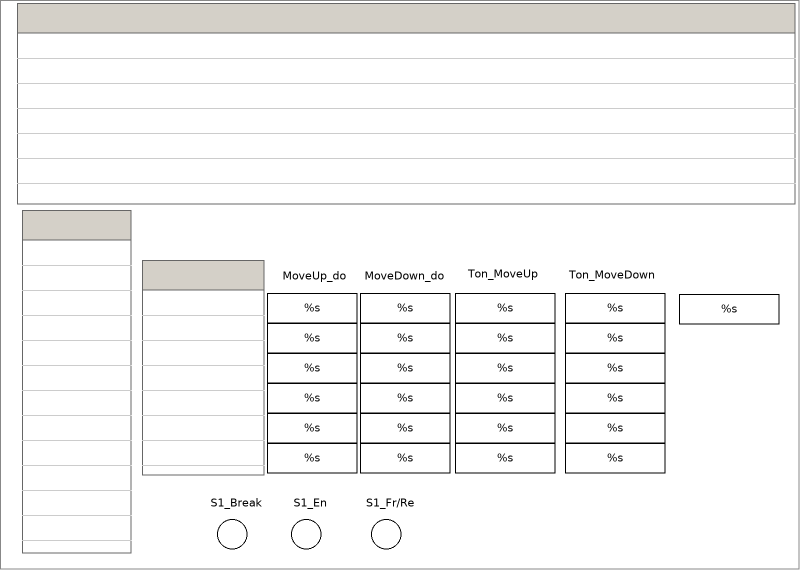
VISUALIZATION VIS_UpDownSlot  // 800x570
    Table (17,3 778x201), data array: GVL_API.stUpDownSlot
        p3854506369: GVL_API.stUpDownSlot[INDEX].error_code
        p1892666644: GVL_API.stUpDownSlot[INDEX].state
        p338671338: GVL_API.stUpDownSlot[INDEX].sensor_up
        p2170511999: GVL_API.stUpDownSlot[INDEX].sensor_down
        p3723444502: GVL_API.stUpDownSlot[INDEX].Error
        p1218418051: GVL_API.stUpDownSlot[INDEX].Initialize
        p746581629: GVL_API.stUpDownSlot[INDEX].MoveDown
        p3104783080: GVL_API.stUpDownSlot[INDEX].MoveUp
        p2501879983: GVL_API.stUpDownSlot[INDEX].Setoff
        p7306298: GVL_API.stUpDownSlot[INDEX].timeout_up
        p1933151965: GVL_API.stUpDownSlot[INDEX].timeout_down
        p3863566920: GVL_API.stUpDownSlot[INDEX].extra_down_time
        p4242324053: extra_time
        Columns.Column.[8].Template: toggle GVL_API.stUpDownSlot[INDEX].Setoff
        Columns.Column.[6].Template: toggle GVL_API.stUpDownSlot[INDEX].MoveDown
        Columns.Column.[10].Template: OnMouseDown: write GVL_API.stUpDownSlot[INDEX].timeout_down via Default
        Columns.Column.[5].Template: toggle GVL_API.stUpDownSlot[INDEX].Initialize
        Columns.Column.[11].Template: OnMouseDown: write GVL_API.stUpDownSlot[INDEX].extra_down_time via Default
        Columns.Column.[7].Template: toggle GVL_API.stUpDownSlot[INDEX].MoveUp
        Columns.Column.[9].Template: OnMouseDown: write GVL_API.stUpDownSlot[INDEX].timeout_up via Default
        Columns.Column.[1].Template: GVL_API.stUpDownSlot[INDEX].state=100
    Rectangle (565,293 100x30), "%s", text variable: P_UpDownSlot.UpDownSlot_S1.Ton_MoveDown_do.ET
    Table (142,260 122x215), data array: stInput.biUDS_sensor_up_S
        p1892666644: stInput.biUDS_sensor[INDEX].sensor_up_right
        p338671338: stInput.biUDS_sensor[INDEX].sensor_down_left
        p2170511999: stInput.biUDS_sensor[INDEX].sensor_down_right
        p3854506369: stInput.biUDS_sensor_up_S[INDEX]
        Columns.Column.[0].Template: toggle stInput.biUDS_sensor_up_S[INDEX]
    Rectangle (565,353 100x30), "%s", text variable: P_UpDownSlot.UpDownSlot_S2_S6[3].Ton_MoveDown_do.ET
    Rectangle (565,383 100x30), "%s", text variable: P_UpDownSlot.UpDownSlot_S2_S6[4].Ton_MoveDown_do.ET
    Rectangle (565,413 100x30), "%s", text variable: P_UpDownSlot.UpDownSlot_S2_S6[5].Ton_MoveDown_do.ET
    Rectangle (565,323 100x30), "%s", text variable: P_UpDownSlot.UpDownSlot_S2_S6[2].Ton_MoveDown_do.ET
    Rectangle (455,293 100x30), "%s", text variable: P_UpDownSlot.UpDownSlot_S1.Ton_MoveUp_do.ET
    Rectangle (455,323 100x30), "%s", text variable: P_UpDownSlot.UpDownSlot_S2_S6[2].Ton_MoveUp_do.ET
    Rectangle (455,353 100x30), "%s", text variable: P_UpDownSlot.UpDownSlot_S2_S6[3].Ton_MoveUp_do.ET
    Rectangle (455,383 100x30), "%s", text variable: P_UpDownSlot.UpDownSlot_S2_S6[4].Ton_MoveUp_do.ET
    Rectangle (455,413 100x30), "%s", text variable: P_UpDownSlot.UpDownSlot_S2_S6[5].Ton_MoveUp_do.ET
    Label (559,260 106x30), "Ton_MoveDown"
    Label (451,259 104x30), "Ton_MoveUp"
    Table (22,210 109x343), data array: stInput.biUDS_sensor_down_S1
        p3854506369: stInput.biUDS_sensor_down_S1[INDEX]
        p1892666644: stInput.biUDS_sensor[INDEX].sensor_up_right
        p338671338: stInput.biUDS_sensor[INDEX].sensor_down_left
        p2170511999: stInput.biUDS_sensor[INDEX].sensor_down_right
        Columns.Column.[0].Template: toggle stInput.biUDS_sensor_down_S1[INDEX]
    Rectangle (565,443 100x30), "%s", text variable: P_UpDownSlot.UpDownSlot_S2_S6[6].Ton_MoveDown_do.ET
    Rectangle (455,443 100x30), "%s", text variable: P_UpDownSlot.UpDownSlot_S2_S6[6].Ton_MoveUp_do.ET
    Rectangle (679,294 100x30), "%s", text variable: P_UpDownSlot.UpDownSlot_S1.Ton_MoveDown_delay_do.ET
    Ellipse (217,519 30x30), colour toggle: stOutput.bqS1_Break
    Label (202,488 69x30), "S1_Break"
    Rectangle (267,323 90x30), "%s", text variable: stOutput.bqUDS_MoveUp_do[2], colour toggle: stOutput.bqUDS_MoveUp_do[2]
    Label (268,261 93x30), "MoveUp_do"
    Rectangle (360,323 90x30), "%s", text variable: stOutput.bqUDS_MoveDown_do[2], colour toggle: stOutput.bqUDS_MoveDown_do[2]
    Label (358,261 93x30), "MoveDown_do"
    Rectangle (267,353 90x30), "%s", text variable: stOutput.bqUDS_MoveUp_do[3], colour toggle: stOutput.bqUDS_MoveUp_do[3]
    Rectangle (267,383 90x30), "%s", text variable: stOutput.bqUDS_MoveUp_do[4], colour toggle: stOutput.bqUDS_MoveUp_do[4]
    Rectangle (267,413 90x30), "%s", text variable: stOutput.bqUDS_MoveUp_do[5], colour toggle: stOutput.bqUDS_MoveUp_do[5]
    Rectangle (267,443 90x30), "%s", text variable: stOutput.bqUDS_MoveUp_do[6], colour toggle: stOutput.bqUDS_MoveUp_do[6]
    Rectangle (360,353 90x30), "%s", text variable: stOutput.bqUDS_MoveDown_do[3], colour toggle: stOutput.bqUDS_MoveDown_do[3]
    Rectangle (360,383 90x30), "%s", text variable: stOutput.bqUDS_MoveDown_do[4], colour toggle: stOutput.bqUDS_MoveDown_do[4]
    Rectangle (360,413 90x30), "%s", text variable: stOutput.bqUDS_MoveDown_do[5], colour toggle: stOutput.bqUDS_MoveDown_do[5]
    Rectangle (360,443 90x30), "%s", text variable: stOutput.bqUDS_MoveDown_do[6], colour toggle: stOutput.bqUDS_MoveDown_do[6]
    Rectangle (267,293 90x30), "%s", text variable: P_UpDownSlot.UpDownSlot_S1.MoveUp_do, colour toggle: P_UpDownSlot.UpDownSlot_S1.MoveUp_do
    Rectangle (360,293 90x30), "%s", text variable: P_UpDownSlot.UpDownSlot_S1.MoveDown_do, colour toggle: P_UpDownSlot.UpDownSlot_S1.MoveDown_do
    Ellipse (291,519 30x30), colour toggle: stOutput.bqS1_Drive_enabled
    Label (276,488 69x30), "S1_En"
    Ellipse (371,519 30x30), colour toggle: stOutput.bqS1_Forward_Reverse
    Label (356,488 69x30), "S1_Fr/Re"
END_VISUALIZATION

(* stored: Version 1.1.0.1, ProductVersion 3.1.4024.11
   Visu VIS_UpDownSlot: Id {1643c897-e951-4b55-b5cf-f408289e75de} *)
